Yaskawa INFORM job: ROS_S1.JBI

/JOB
//NAME ROS_S1
//POS
///NPOS 0,0,0,0,0,0
//INST
///DATE 2016/01/14 15:24
///ATTR SC,RW
///GROUP1 ST1
NOP
TIMER T=0.05
SKILLSND SL6 "ROS-START"
TSYNC 1
WAIT OT#(890)=ON
SKILLSND SL6 "ROS-STOP"
END
